(* IEC 61131-3 sources: PLC-Obfuscation/templates, 3 files *)

(* ---- random_f_snap.st ---- *)
FUNCTION_BLOCK rand_generator
  VAR_INPUT
    IN : BOOL;
  END_VAR
  VAR
    M : BOOL := 0;
    INIT : BOOL := 0;
  END_VAR
  VAR_OUTPUT
    OUT : INT := 0;
  END_VAR

  (* Initialize our random generator *)
  (* This IF is called only the first time this *)
  (* block executes *)
  IF INIT = 0 THEN
    {
    srand(17);}
    INIT := 1;
  END_IF;

  IF M = 0 and IN = 1 THEN
    (* Using pragma to write code directly in C. *)
    (* You can access your PLC program variables using *)
    (* GetFbVar(var,...) and SetFbVar(var,val,...) calls *)
    {SetFbVar(OUT,  rand() % 1000 )}

  END_IF;
  M := IN;
END_FUNCTION_BLOCK

(* ---- periodic_snap.st ---- *)
  VAR
    current_time_internal AT %ML1024 : ULINT;
  END_VAR
  VAR
    obf_p: INT := ${period};
    obf_tmp: INT;
	obf_t: INT;
  END_VAR
  VAR
 	${new_var} AT %${new_reg}: BOOL;
  END_VAR

  obf_t := ABS(LWORD_TO_INT( AND( LINT_TO_LWORD(2147483647), ULINT_TO_LWORD(current_time_internal) ) ));
  obf_tmp := MOD(obf_t, obf_p);
  ${new_var} := LE(obf_tmp, DIV(obf_p,2));

(* ---- random_snap.st ---- *)
  VAR
     obf_r: INT := 100;
   END_VAR
  VAR
   	${new_var} AT %${new_reg}: BOOL;
  END_VAR
  VAR
    obf_ra : BOOL;
  END_VAR
  VAR
    rand_generator0 : rand_generator;
  END_VAR

  rand_generator0(IN := ${dep_register});
  obf_ra := LE(rand_generator0.OUT, obf_r);
  ${new_var} := NOT(${new_var}) AND obf_ra;
